// TIA Portal V17 export
// export: Created 2025-03-07T09:18:33.1725416Z, ExportSetting WithDefaults, DisplayName Totally Integrated Automation Portal, DisplayVersion V17 Update 8, DisplayName TIA Portal Openness, DisplayVersion V17 Update 8, DisplayName TIA Portal Version Control Interface, DisplayVersion V17, DisplayName SINAMICS Startdrive Advanced, DisplayVersion V17 SP2, DisplayName SINAMICS Startdrive G110M, G120, G120C, G120D, G120P, G115D, DisplayVersion V17 SP2, DisplayName SINAMICS Startdrive G130, G150, S120, S150, SINAMICS MV, S210, DisplayVersion V17 SP2, DisplayName STEP 7 Professional, DisplayVersion V17 Update 8, DisplayName SINUMERIK ONE STEP 7 Toolbox, DisplayVersion V17 Update 12, DisplayName SINUMERIK 840D sl STEP 7 Toolbox, DisplayVersion V17 Update 12, DisplayName STEP 7 Safety, DisplayVersion V17 Update 6, DisplayName WinCC Advanced, DisplayVersion V17 Update 8
DATA_BLOCK "UPTL_ExternalWorkpieceData"   // DB1052
TITLE = UPTL_ExternalWorkpieceData
{ S7_Optimized_Access := 'FALSE'; DB_Accessible_From_OPC_UA := 'FALSE' }
AUTHOR : Transline
FAMILY : TRANSLINE_SINUMERIK-ONE
VERSION : 4.0
// Example for an external workpiece counter DB / Beispiel für einen externen Werkstückzähler-DB
// stored: AutoNumber true, DBAccessibleFromOPCUA false, DBAccessibleFromWebserver true, IsOnlyStoredInLoadMemory false, IsWriteProtectedInAS false
   VAR RETAIN
      CounterOfWorkpieceType { S7_SetPoint := 'True'} : Array[33..34] of "LTLP_typeWorkpieceCount";   // Zählwerte für Werkstücktypen mit Index > 32 in Typvorwahl definierten / Define count values for workpiece types with index > 32 in type preselection
   END_VAR
BEGIN
END_DATA_BLOCK
